(*	Sample Code Disclaimer
	All sample code provided by Beckhoff Automation LLC are for illustrative purposes only
	and are provided “as is” and without any warranties, express or implied.
	Actual implementations in applications will vary significantly.
	Beckhoff Automation LLC shall have no liability for, and does not waive any rights in relation to,
	any code samples that it provides or the use of such code samples for any purpose.
*)
PROGRAM MAIN
VAR
	Machine: FB_UM_Machine	:= (Name := 'Machine', LogStateChanges := TRUE);
	Initialized: BOOL;
END_VAR

CyclicLogic();

METHOD CyclicLogic : BOOL
VAR_INPUT
END_VAR
IF NOT Initialized THEN
    Initialized := Initialize();
    RETURN;
END_IF

Machine.CyclicLogic();
END_METHOD

METHOD Initialize : BOOL
VAR_INPUT
END_VAR
Initialize := TRUE;
END_METHOD

END_PROGRAM

(* stored: Version 1.1.0.1, ProductVersion 3.1.4024.12
   POU MAIN: Id {45fee981-a966-4811-959d-34a789337a55}, SpecialFunc None
   Method CyclicLogic: Id {fe332985-0e52-4a1e-a556-33a8822260d7}
   Method Initialize: Id {b3cc5d6e-29f4-4149-9705-156e78b671c1} *)
